INTERFACE IPistonGripper

METHOD Close : TcoCore.ITcoTaskStatus
END_METHOD

METHOD Open : TcoCore.ITcoTaskStatus
END_METHOD

END_INTERFACE

(* stored: Version 1.1.0.1
   Itf IPistonGripper: Id {ccfb8387-bc57-0c8d-2774-5d93bca1f648}
   Folder Gripper: Id {876b84e8-9533-0895-3053-8d7d5f87e8c2}
   Method Close: Id {f5b26b0b-7fa2-0f10-3599-0e58033f47d2}
   Method Open: Id {6be07815-b97a-01f3-343f-f606e4492b30} *)
